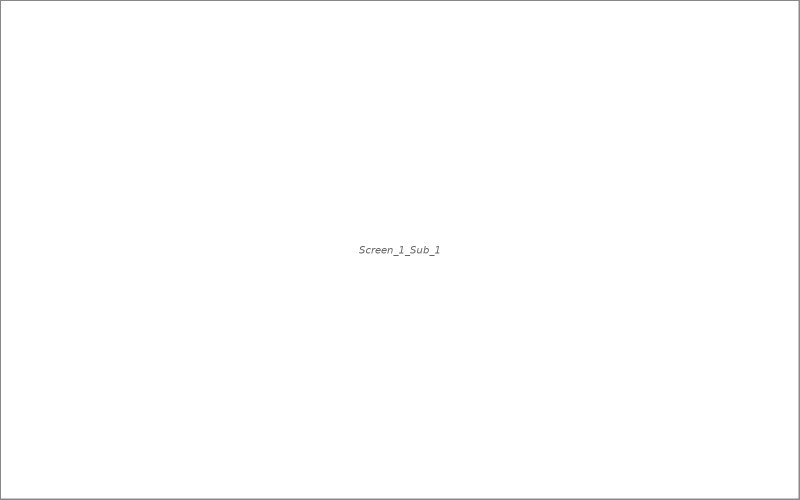
VISUALIZATION Screen_1  // 800x500
    TabControl (0,0 800x500)
        shows Screen_1_Sub_1()
        shows Screen_1_Sub_2()
        shows Screen_1_Sub_3()
        shows Screen_1_Sub_4()
        [0]: TabTitle=Tombol Valve
        [1]: TabTitle=Digital Input
        [2]: TabTitle=Num Display 1
        [3]: TabTitle=Num Display 2
END_VISUALIZATION

(* stored: Version 1.1.0.1, ProductVersion 3.1.4024.12
   Visu Screen_1: Id {068bc64c-15f2-4039-90c6-6906f1d1b752} *)
